RoboDK station: wcs_plc_20240203_183935.rdk

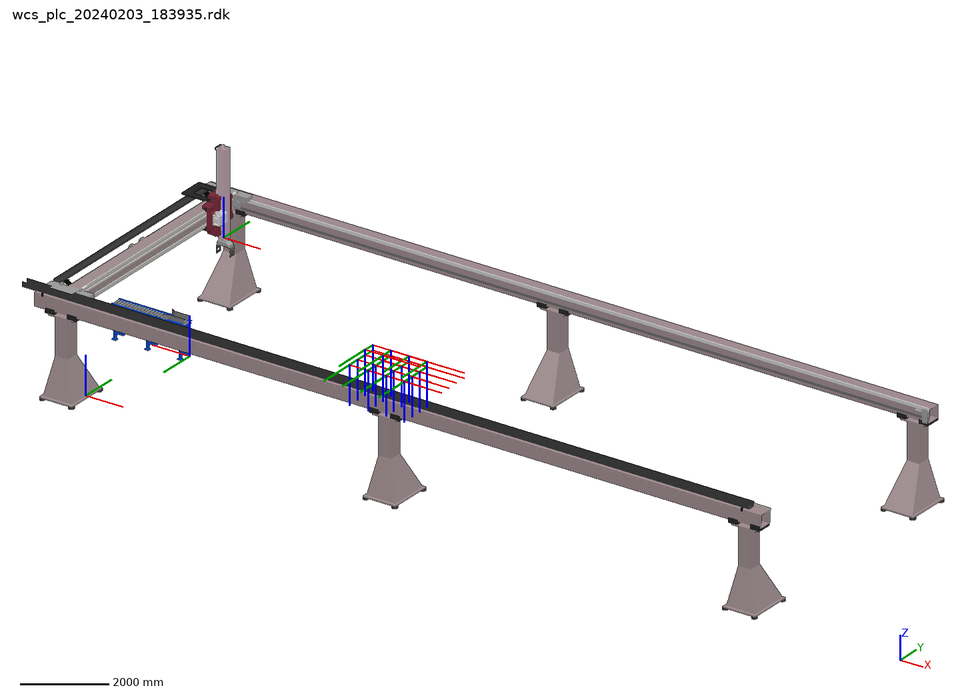
[picture v0: the station drawn from its stored meshes, robots at their saved joint values, targets as dots, program paths as lines]
Station init (saved by RoboDK 5.6.8). Poses are relative to the parent item; angles as X-Y-Z fixed-axis rotations.
Station parameters (name, value as stored): TAGS, ['Milling']
  - frame conveyor Base at (750, 3000, 0) mm, rotated rx 0 ry 0 rz 180 deg
    - robot conveyor: 1 axes
        modified DH rows (alpha deg, a mm, theta deg, d mm): 0, 0, 0, 0 linear
        base shift (0, 0, 0) mm, rotated rx 0 ry 90 rz 0 deg
        joint limits [-99999] to [9999999]; home [0]; saved at [1000]
      - tool conveyor_TCP, TCP at (160, 110, 135) mm, rotated rx -180 ry 0 rz -180 deg
    - target con_pitch (joint target) at (1000, 0, 880) mm; joints [1000, 0, 0] of conveyor
    - target con_home (joint target) at (160, 110, 1015) mm, rotated rx -180 ry 0 rz -180 deg; joints [0] of conveyor
  - frame gantry Base at (0, 0, 0) mm
    - robot gantry: 3 axes
        modified DH rows (alpha deg, a mm, theta deg, d mm): 0, 0, 0, 0 linear; 90, 0, 90, 0 linear; 90, 0, 0, 0 linear
        base shift (0, 0, 0) mm, rotated rx 0 ry -90 rz 180 deg
        joint limits [-5, -5, -5] to [18000, 5000, 1500]; home [0, 0, 0]; saved at [0, 0, 0]
      - frame gripper Base at (0, 0, 0) mm, rotated rx -180 ry 0 rz 0 deg
        - robot gripper: 1 axes
            modified DH rows (alpha deg, a mm, theta deg, d mm): 0, 0, 0, 0 linear
            base shift (0, 0, 0) mm, rotated rx 0 ry 90 rz 0 deg
            joint limits [-200] to [0]; home [0]; saved at [0]
        - target close_gripper (joint target) at (-121.33, 5507.34, 1743.56) mm; joints [-55] of gripper
        - target open_gripper (joint target) at (0, 0, 0) mm; joints [0, 0, 0] of gripper
      - tool gripper_TCP, TCP at (0, 0, 260) mm
    - target gantry_home (joint target) at (-66.33, 5507.34, 1483.56) mm, rotated rx 180 ry 0 rz 0 deg; joints [0, 0, 0] of gantry
    - target UP_pickup (joint target) at (590, 2890, 1483.56) mm, rotated rx 180 ry 0 rz 0 deg; joints [656.33, 2617.342, 0] of gantry
    - target IN_pickup (joint target) at (590, 2890, 1015) mm, rotated rx 180 ry 0 rz 0 deg; joints [656.33, 2617.342, 468.564] of gantry
    - target Target 6 (joint target) at (4133.67, 4957.34, 433.56) mm, rotated rx 180 ry 0 rz 0 deg; joints [4200, 550, 1050] of gantry
    - target Target 7 (Cartesian target) at (10933.67, 1007.34, 433.56) mm, rotated rx 180 ry 0 rz 0 deg; joints [11000, 4500, 1050] of gantry
    - folder pallet
      - frame TeachingPoints_01-01-01 at (4633.67, 4657.34, 568.56) mm, rotated rx 180 ry 0 rz 0 deg
        - target Point_01-01-01 (Cartesian target) at (0, 0, 0) mm; joints [4700, 850, 915] of gantry
      - frame TeachingPoints_02-01-01 at (5133.67, 4657.34, 568.56) mm, rotated rx 180 ry 0 rz 0 deg
        - target Point_02-01-01 (Cartesian target) at (0, 0, 0) mm; joints [5200, 850, 915] of gantry
      - frame TeachingPoints_03-01-01 at (5633.67, 4657.34, 568.56) mm, rotated rx 180 ry 0 rz 0 deg
        - target Point_03-01-01 (Cartesian target) at (0, 0, 0) mm; joints [5700, 850, 915] of gantry
      - frame TeachingPoints_04-01-01 at (6133.67, 4657.34, 568.56) mm, rotated rx 180 ry 0 rz 0 deg
        - target Point_04-01-01 (Cartesian target) at (0, 0, 0) mm; joints [6200, 850, 915] of gantry
      - frame TeachingPoints_01-02-01 at (4633.67, 4357.34, 568.56) mm, rotated rx 180 ry 0 rz 0 deg
        - target Point_01-02-01 (Cartesian target) at (0, 0, 0) mm; joints [4700, 1150, 915] of gantry
      - frame TeachingPoints_02-02-01 at (5133.67, 4357.34, 568.56) mm, rotated rx 180 ry 0 rz 0 deg
        - target Point_02-02-01 (Cartesian target) at (0, 0, 0) mm; joints [5200, 1150, 915] of gantry
      - frame TeachingPoints_03-02-01 at (5633.67, 4357.34, 568.56) mm, rotated rx 180 ry 0 rz 0 deg
        - target Point_03-02-01 (Cartesian target) at (0, 0, 0) mm; joints [5700, 1150, 915] of gantry
      - frame TeachingPoints_04-02-01 at (6133.67, 4357.34, 568.56) mm, rotated rx 180 ry 0 rz 0 deg
        - target Point_04-02-01 (Cartesian target) at (0, 0, 0) mm; joints [6200, 1150, 915] of gantry
      - frame TeachingPoints_01-03-01 at (4633.67, 4057.34, 568.56) mm, rotated rx 180 ry 0 rz 0 deg
        - target Point_01-03-01 (Cartesian target) at (0, 0, 0) mm; joints [4700, 1450, 915] of gantry
      - frame TeachingPoints_02-03-01 at (5133.67, 4057.34, 568.56) mm, rotated rx 180 ry 0 rz 0 deg
        - target Point_02-03-01 (Cartesian target) at (0, 0, 0) mm; joints [5200, 1450, 915] of gantry
      - frame TeachingPoints_03-03-01 at (5633.67, 4057.34, 568.56) mm, rotated rx 180 ry 0 rz 0 deg
        - target Point_03-03-01 (Cartesian target) at (0, 0, 0) mm; joints [5700, 1450, 915] of gantry
      - frame TeachingPoints_04-03-01 at (6133.67, 4057.34, 568.56) mm, rotated rx 180 ry 0 rz 0 deg
        - target Point_04-03-01 (Cartesian target) at (0, 0, 0) mm; joints [6200, 1450, 915] of gantry
      - frame TeachingPoints_01-04-01 at (4633.67, 3757.34, 568.56) mm, rotated rx 180 ry 0 rz 0 deg
        - target Point_01-04-01 (Cartesian target) at (0, 0, 0) mm; joints [4700, 1750, 915] of gantry
      - frame TeachingPoints_02-04-01 at (5133.67, 3757.34, 568.56) mm, rotated rx 180 ry 0 rz 0 deg
        - target Point_02-04-01 (Cartesian target) at (0, 0, 0) mm; joints [5200, 1750, 915] of gantry
      - frame TeachingPoints_03-04-01 at (5633.67, 3757.34, 568.56) mm, rotated rx 180 ry 0 rz 0 deg
        - target Point_03-04-01 (Cartesian target) at (0, 0, 0) mm; joints [5700, 1750, 915] of gantry
      - frame TeachingPoints_04-04-01 at (6133.67, 3757.34, 568.56) mm, rotated rx 180 ry 0 rz 0 deg
        - target Point_04-04-01 (Cartesian target) at (0, 0, 0) mm; joints [6200, 1750, 915] of gantry
      - frame TeachingPoints_01-01-02 at (4633.67, 4657.34, 703.56) mm, rotated rx 180 ry 0 rz 0 deg
        - target Point_01-01-02 (Cartesian target) at (0, 0, 0) mm; joints [4700, 850, 780] of gantry
      - frame TeachingPoints_02-01-02 at (5133.67, 4657.34, 703.56) mm, rotated rx 180 ry 0 rz 0 deg
        - target Point_02-01-02 (Cartesian target) at (0, 0, 0) mm; joints [5200, 850, 780] of gantry
      - frame TeachingPoints_03-01-02 at (5633.67, 4657.34, 703.56) mm, rotated rx 180 ry 0 rz 0 deg
        - target Point_03-01-02 (Cartesian target) at (0, 0, 0) mm; joints [5700, 850, 780] of gantry
      - frame TeachingPoints_04-01-02 at (6133.67, 4657.34, 703.56) mm, rotated rx 180 ry 0 rz 0 deg
        - target Point_04-01-02 (Cartesian target) at (0, 0, 0) mm; joints [6200, 850, 780] of gantry
      - frame TeachingPoints_01-02-02 at (4633.67, 4357.34, 703.56) mm, rotated rx 180 ry 0 rz 0 deg
        - target Point_01-02-02 (Cartesian target) at (0, 0, 0) mm; joints [4700, 1150, 780] of gantry
      - frame TeachingPoints_02-02-02 at (5133.67, 4357.34, 703.56) mm, rotated rx 180 ry 0 rz 0 deg
        - target Point_02-02-02 (Cartesian target) at (0, 0, 0) mm; joints [5200, 1150, 780] of gantry
      - frame TeachingPoints_03-02-02 at (5633.67, 4357.34, 703.56) mm, rotated rx 180 ry 0 rz 0 deg
        - target Point_03-02-02 (Cartesian target) at (0, 0, 0) mm; joints [5700, 1150, 780] of gantry
      - frame TeachingPoints_04-02-02 at (6133.67, 4357.34, 703.56) mm, rotated rx 180 ry 0 rz 0 deg
        - target Point_04-02-02 (Cartesian target) at (0, 0, 0) mm; joints [6200, 1150, 780] of gantry
      - frame TeachingPoints_01-03-02 at (4633.67, 4057.34, 703.56) mm, rotated rx 180 ry 0 rz 0 deg
        - target Point_01-03-02 (Cartesian target) at (0, 0, 0) mm; joints [4700, 1450, 780] of gantry
      - frame TeachingPoints_02-03-02 at (5133.67, 4057.34, 703.56) mm, rotated rx 180 ry 0 rz 0 deg
        - target Point_02-03-02 (Cartesian target) at (0, 0, 0) mm; joints [5200, 1450, 780] of gantry
      - frame TeachingPoints_03-03-02 at (5633.67, 4057.34, 703.56) mm, rotated rx 180 ry 0 rz 0 deg
        - target Point_03-03-02 (Cartesian target) at (0, 0, 0) mm; joints [5700, 1450, 780] of gantry
      - frame TeachingPoints_04-03-02 at (6133.67, 4057.34, 703.56) mm, rotated rx 180 ry 0 rz 0 deg
        - target Point_04-03-02 (Cartesian target) at (0, 0, 0) mm; joints [6200, 1450, 780] of gantry
      - frame TeachingPoints_01-04-02 at (4633.67, 3757.34, 703.56) mm, rotated rx 180 ry 0 rz 0 deg
        - target Point_01-04-02 (Cartesian target) at (0, 0, 0) mm; joints [4700, 1750, 780] of gantry
      - frame TeachingPoints_02-04-02 at (5133.67, 3757.34, 703.56) mm, rotated rx 180 ry 0 rz 0 deg
        - target Point_02-04-02 (Cartesian target) at (0, 0, 0) mm; joints [5200, 1750, 780] of gantry
      - frame TeachingPoints_03-04-02 at (5633.67, 3757.34, 703.56) mm, rotated rx 180 ry 0 rz 0 deg
        - target Point_03-04-02 (Cartesian target) at (0, 0, 0) mm; joints [5700, 1750, 780] of gantry
      - frame TeachingPoints_04-04-02 at (6133.67, 3757.34, 703.56) mm, rotated rx 180 ry 0 rz 0 deg
        - target Point_04-04-02 (Cartesian target) at (0, 0, 0) mm; joints [6200, 1750, 780] of gantry
  - frame Frame 36 at (12000, 3370, 2800) mm, rotated rx -105 ry 0 rz 90 deg
  - camera Camera 1
